// Mitsubishi GX Works2 project: YKHMI-Fx1s-XY-v1.0   PLC: FX1S

PROGRAM MAIN
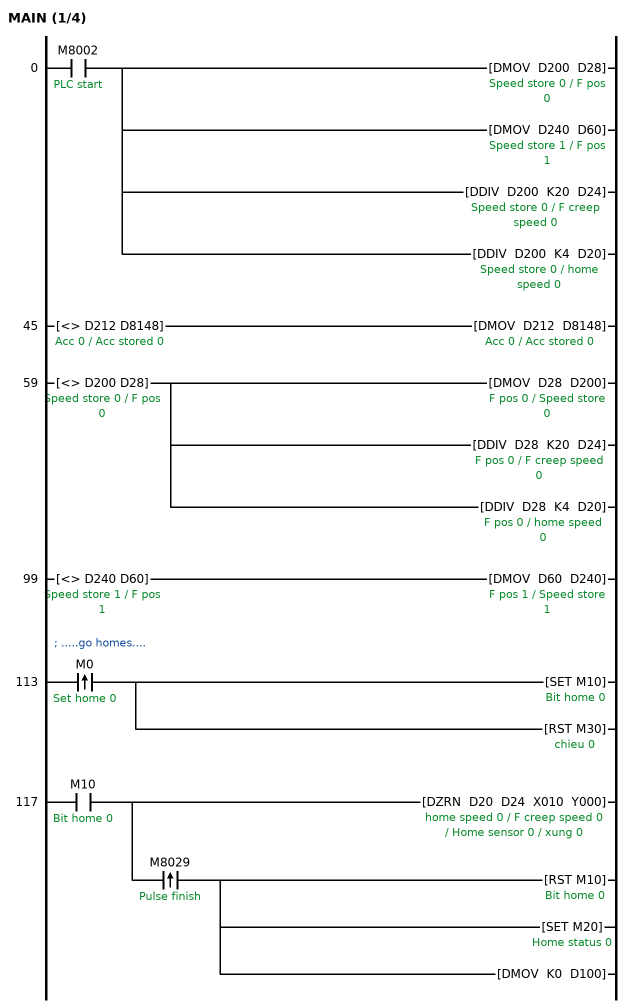
0     LD      M8002  ; PLC start
      DMOV    D200 D28  ; Speed store 0 / F pos 0
      DMOV    D240 D60  ; Speed store 1 / F pos 1
      DDIV    D200 K20 D24  ; F creep speed 0
      DDIV    D200 K4 D20  ; home speed 0
45    LD<>    D212 D8148  ; Acc 0 / Acc stored 0
      DMOV    D212 D8148
59    LD<>    D200 D28  ; Speed store 0 / F pos 0
      DMOV    D28 D200
      DDIV    D28 K20 D24
      DDIV    D28 K4 D20
99    LD<>    D240 D60  ; Speed store 1 / F pos 1
      DMOV    D60 D240
; .....go homes....
113   LDP     M0  ; Set home 0
      SET     M10  ; Bit home 0
      RST     M30  ; chieu 0
117   LD      M10  ; Bit home 0
      DZRN    D20 D24 X010 Y000  ; Home sensor 0 / xung 0
      ANDP    M8029  ; Pulse finish
      RST     M10  ; Bit home 0
      SET     M20  ; Home status 0
      DMOV    K0 D100
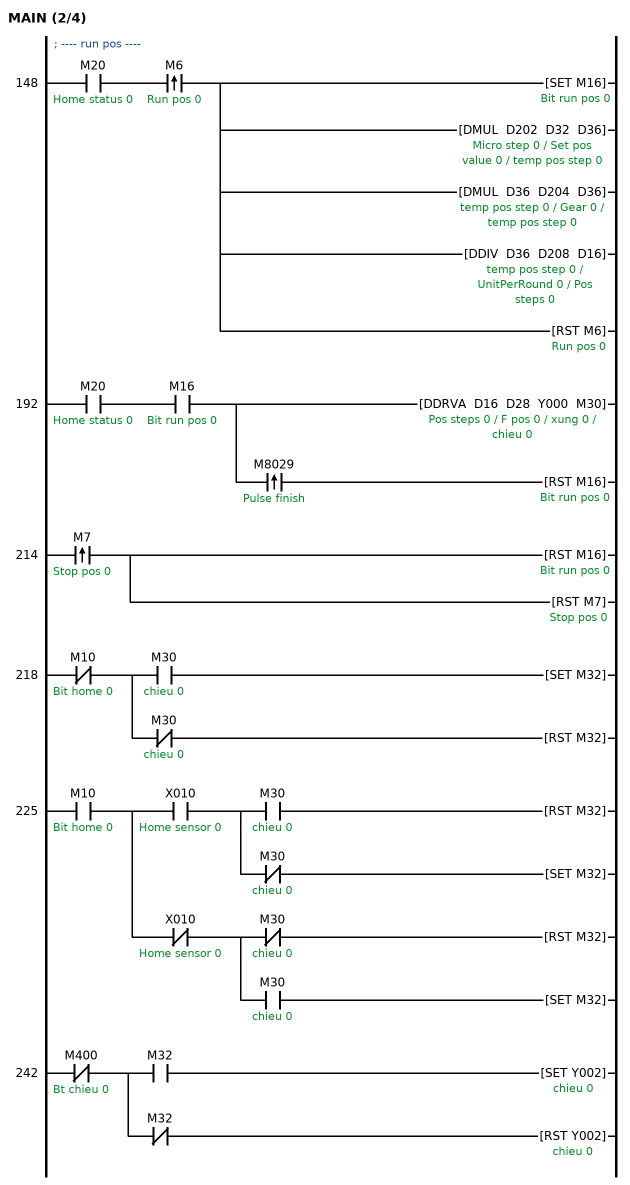
; ---- run pos ----
148   LD      M20  ; Home status 0
      ANDP    M6  ; Run pos 0
      SET     M16  ; Bit run pos 0
      DMUL    D202 D32 D36  ; Micro step 0 / Set pos value 0 / temp pos step 0
      DMUL    D36 D204 D36  ; Gear 0
      DDIV    D36 D208 D16  ; UnitPerRound 0 / Pos steps 0
      RST     M6  ; Run pos 0
192   LD      M20  ; Home status 0
      AND     M16  ; Bit run pos 0
      DDRVA   D16 D28 Y000 M30
      ANDP    M8029  ; Pulse finish
      RST     M16  ; Bit run pos 0
214   LDP     M7  ; Stop pos 0
      RST     M16  ; Bit run pos 0
      RST     M7  ; Stop pos 0
; 
218   LDI     M10  ; Bit home 0
      MPS
      AND     M30  ; chieu 0
      SET     M32
      MPP
      ANI     M30  ; chieu 0
      RST     M32
225   LD      M10  ; Bit home 0
      MPS
      AND     X010  ; Home sensor 0
      MPS
      AND     M30  ; chieu 0
      RST     M32
      MPP
      ANI     M30  ; chieu 0
      SET     M32
      MPP
      ANI     X010  ; Home sensor 0
      MPS
      ANI     M30  ; chieu 0
      RST     M32
      MPP
      AND     M30  ; chieu 0
      SET     M32
242   LDI     M400  ; Bt chieu 0
      MPS
      AND     M32
      SET     Y002  ; chieu 0
      MPP
      ANI     M32
      RST     Y002  ; chieu 0
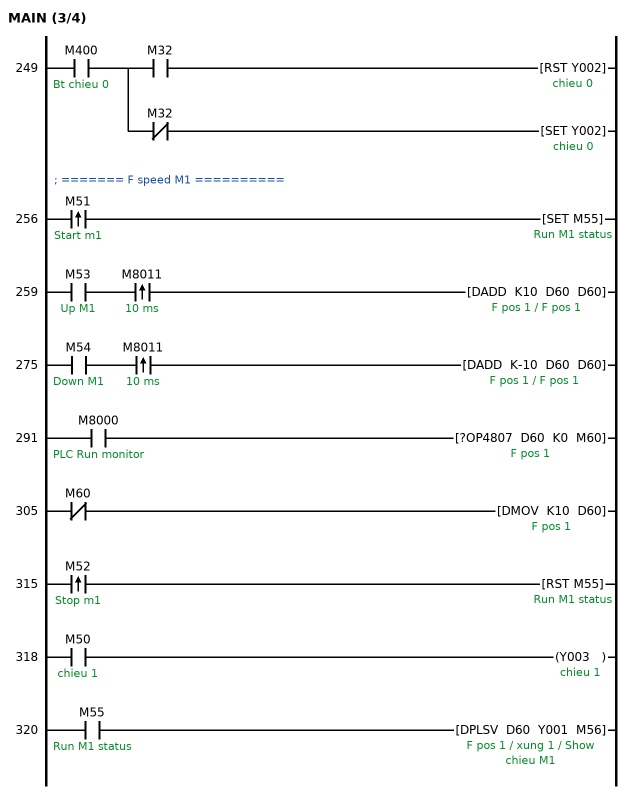
249   LD      M400  ; Bt chieu 0
      MPS
      AND     M32
      RST     Y002  ; chieu 0
      MPP
      ANI     M32
      SET     Y002  ; chieu 0
; ======= F speed M1 ==========
256   LDP     M51  ; Start m1
      SET     M55  ; Run M1 status
259   LD      M53  ; Up M1
      ANDP    M8011  ; 10 ms
      DADD    K10 D60 D60
275   LD      M54  ; Down M1
      ANDP    M8011  ; 10 ms
      DADD    K-10 D60 D60
291   LD      M8000  ; PLC Run monitor
      ?OP4807 D60 K0 M60
305   LDI     M60
      DMOV    K10 D60
315   LDP     M52  ; Stop m1
      RST     M55  ; Run M1 status
318   LD      M50  ; chieu 1
      OUT     Y003  ; chieu 1
320   LD      M55  ; Run M1 status
      DPLSV   D60 Y001 M56  ; xung 1 / Show chieu M1
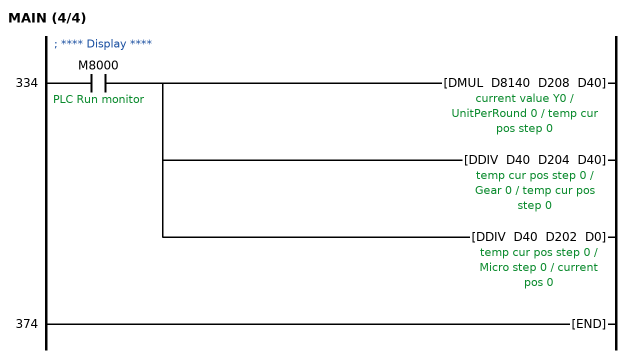
; **** Display ****
334   LD      M8000  ; PLC Run monitor
      DMUL    D8140 D208 D40  ; current value Y0 / temp cur pos step 0
      DDIV    D40 D204 D40
      DDIV    D40 D202 D0  ; current pos 0
374   END
END_PROGRAM

// device comments not shown above
M1  ; jog + 0
Y014  ; en 0 & 1
Y015  ; Out xilanh
M2  ; jog- 0
M3  ; F forward 0
M4  ; F reverse 0
M5  ; Stop jog 0
M8  ; Stop F 0
M9  ; Run AB 0
M11  ; Bit jog+ 0
M12  ; Bit jog- 0
M13  ; BitF forward 0
M14  ; Bit F reverse 0
M17  ; Bit stop pos 0
M18  ; Bit F stop 0
M19  ; Bit Run AB 0
M29  ; Stop AB
M31  ; enable 0
M100  ; Limit position
M101  ; Limit position+
M106  ; Limit pos -
M110  ; Bit cmp > speed
M111  ; Bit cmp = speed
M112  ; Bit cmp < speed
M120  ; Bit cmp run speed and temp speed
M125  ; Bit cmp speed and zero
D4  ; F speed 0
D8  ; Set jog value 0
D12  ; Jog steps 0
D44  ; F speed acc temp 0
D48  ; F speed acc inc 0
D52  ; F speed acc 0
D68  ; DECO run AB
D72  ; Temp delay AB
D206  ; Pos value 0-0
D210  ; N-teeth 0
D220  ; PosA
D222  ; PosB
D224  ; Delay AB
X002  ; Limit- 0
X003  ; Limit+ 0
X004  ; Limit- 1
X005  ; Limit+ 1
X006  ; Xilanh trigger
X011  ; Home sensor 1
